(* Schneider Machine Expert - Basic project PRIMEIRO PROJETO, file version 2.7.0.0 *)
(* ProjectInformations: Name=Novo projeto *)

HARDWARE
  Cpu 0: TM221CE24R
  EthernetConfiguration: NetworkName=M221, IpAllocationMode=FixedAddress, IpAddress=0.0.0.0, SubnetMask=0.0.0.0
  SerialLineConfiguration: Baud=Baud19200, Parity=ParityEven, DataBits=DataBits8, StopBits=StopBits1, PhysicalMedium=PhysicalMediumRs485, TransmissionMode=TransmissionModeModbusRtu, SlaveId=1, Addressing=SlaveAddressing
  MastTask: UsePeriodScanMode=false, PeriodScan=100
  FastTask: Period=255
  CpuBehavior: StartingMode=StartAsPreviousState, AutoSaveRamOnEeprom=true, WatchdogPeriod=250

SYMBOLS  (address, symbol, comment, settings)
  %M10      START_ESTEIRA
  %M11      STOP_ESTEIRA
  %M12      SENSOR_ENTRADA
  %M13      SENSOR_SAIDA
  %M14      SENSOR_CONTADOR
  %M15      RESET_CONTADOR
  %M20      ESTEIRA_INICIO
  %M21      ESTEIRA_FINAL
  %M22      LED_PAUSE
  %M23      LED_START_ESTEIRA
  %M24      LED_STOP_ESTEIRA
  %M25      LED_VERDE
  %M26      EMISSOR
  %M27      LED_VERMELHO
  %M28      LED_AMARELO

POU Novo POU
  (* SectionNumber=1 *)

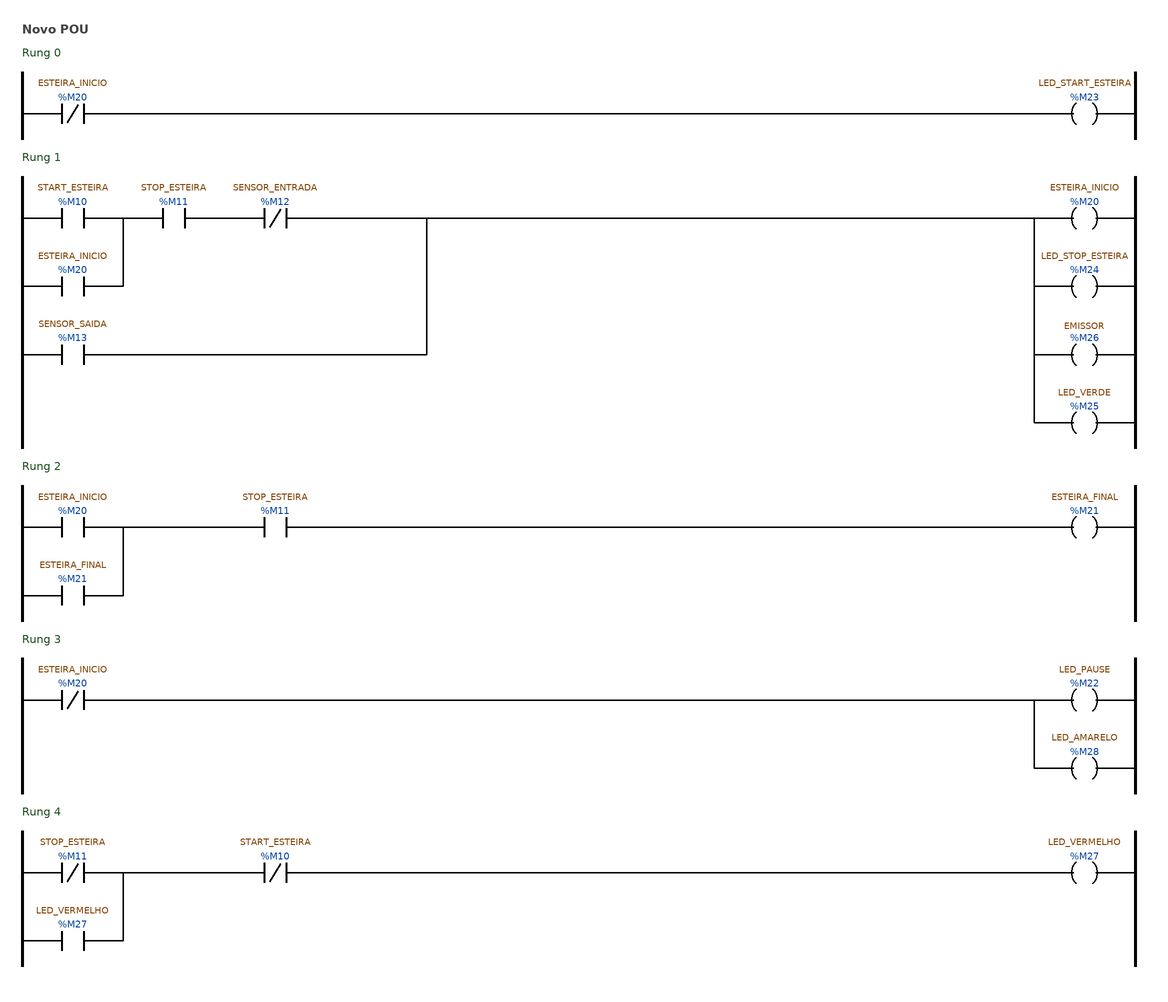

// Rung 0
  LDN %M20                (* ESTEIRA_INICIO *)
  ST %M23                 (* LED_START_ESTEIRA *)
  // as ST:
  //   LED_START_ESTEIRA := NOT ESTEIRA_INICIO;

// Rung 1
  LD %M10                 (* START_ESTEIRA *)
  OR %M20                 (* ESTEIRA_INICIO *)
  AND %M11                (* STOP_ESTEIRA *)
  ANDN %M12               (* SENSOR_ENTRADA *)
  OR %M13                 (* SENSOR_SAIDA *)
  ST %M20                 (* ESTEIRA_INICIO *)
  ST %M24                 (* LED_STOP_ESTEIRA *)
  ST %M26                 (* EMISSOR *)
  ST %M25                 (* LED_VERDE *)
  // as ST:
  //   _t1 := (START_ESTEIRA OR ESTEIRA_INICIO) AND STOP_ESTEIRA AND NOT SENSOR_ENTRADA OR SENSOR_SAIDA;
  //   ESTEIRA_INICIO := _t1;
  //   LED_STOP_ESTEIRA := _t1;
  //   EMISSOR := _t1;
  //   LED_VERDE := _t1;

// Rung 2
  LD %M20                 (* ESTEIRA_INICIO *)
  OR %M21                 (* ESTEIRA_FINAL *)
  AND %M11                (* STOP_ESTEIRA *)
  ST %M21                 (* ESTEIRA_FINAL *)
  // as ST:
  //   ESTEIRA_FINAL := (ESTEIRA_INICIO OR ESTEIRA_FINAL) AND STOP_ESTEIRA;

// Rung 3
  LDN %M20                (* ESTEIRA_INICIO *)
  ST %M22                 (* LED_PAUSE *)
  ST %M28                 (* LED_AMARELO *)
  // as ST:
  //   LED_PAUSE := NOT ESTEIRA_INICIO;
  //   LED_AMARELO := NOT ESTEIRA_INICIO;

// Rung 4
  LDN %M11                (* STOP_ESTEIRA *)
  OR %M27                 (* LED_VERMELHO *)
  ANDN %M10               (* START_ESTEIRA *)
  ST %M27                 (* LED_VERMELHO *)
  // as ST:
  //   LED_VERMELHO := (NOT STOP_ESTEIRA OR LED_VERMELHO) AND NOT START_ESTEIRA;

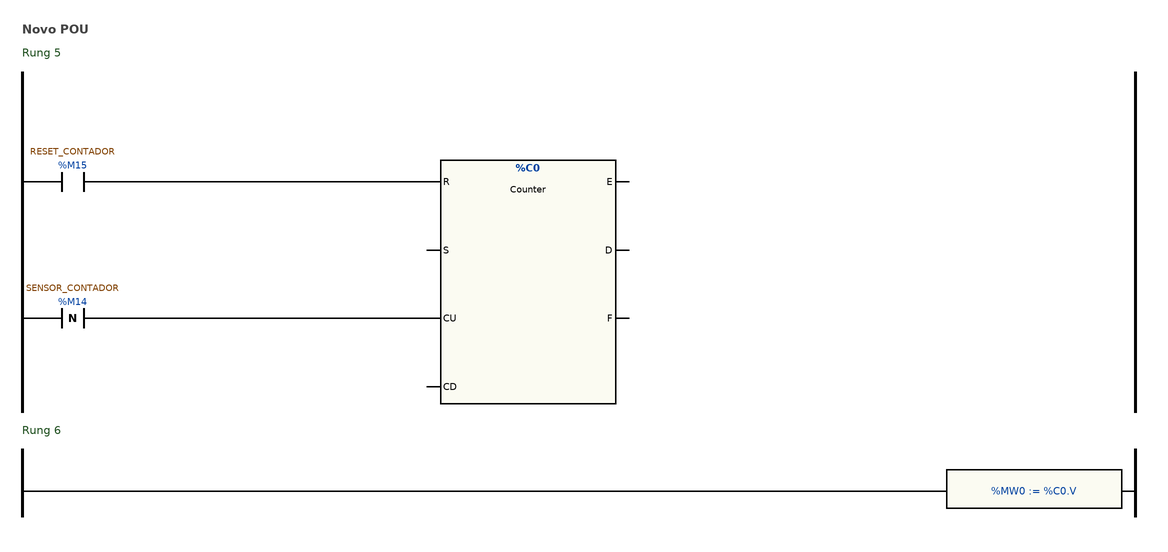

// Rung 5
  BLK %C0
  LD %M15                 (* RESET_CONTADOR *)
  R
  LDF %M14                (* SENSOR_CONTADOR *)
  CU
  END_BLK
  // as ST:
  //   %C0(R := RESET_CONTADOR, CU := FALLING(SENSOR_CONTADOR));

// Rung 6
  LD 1
  [ %MW0 := %C0.V ]
  // as ST:
  //   %MW0 := %C0.V;
